(* IEC 61131-3 sources: eCockpitGit/test_project/src/%F%00 Library/%F%Common Functions/%F%Conversion/%F%Array/%F%BOOL Array, 4 files *)

(* ---- %POU%FU_BoolArrayToDWord.st ---- *)
//This functions converts an array of bools to a word, a maximum of 32 bools can be converted
//It must be used in the following way
//FU_BoolArrayToDWord(pArray:= ADR(BoolArray), usiSize:= SIZEOF(BoolArray));
// |**Version**|**Author**| **Date** |**Changes**
// | 1         | NSN      | 28-03-18 | Creation
// | 1.1       | NSN      | 13-06-18 | Updated names and types
FUNCTION FU_BoolArrayToDWord : DWORD
VAR_INPUT
	pArray			:POINTER TO BOOL;	//Address of bool array
	usiSize			:USINT;				//Size of bool array
END_VAR
VAR
	i				:BYTE;
END_VAR
(*%!%__DELIMITER__%!%*)
IF NOT(usiSize = 0) THEN		//Array must be bigger than 0
	IF usiSize > 32 THEN		//Array must be 32 bools or less
		usiSize				:=		32;
	END_IF
	FOR i := 0 TO usiSize - 1 DO
		FU_dwBitSet(dbVar:=FU_BoolArrayToDWord,bIndex:=i,xVal:=pArray^);
		pArray				:=		pArray + 1;
	END_FOR
END_IF

(* ---- %POU%FU_BoolArrayToWord.st ---- *)
//This functions converts an array of bools to a word, a maximum of 16 bools can be converted
//It must be used in the following way
//FU_BoolArrayToWord(pArray:= ADR(BoolArray), usiSize:= SIZEOF(BoolArray));
// |**Version**|**Author**| **Date** |**Changes**
// | 1         | NSN      | 08-03-18 | Creation
// | 1.1       | NSN      | 13-06-18 | Updated names and types
FUNCTION FU_BoolArrayToWord : WORD
VAR_INPUT
	pArray			:POINTER TO BOOL;	//Address of bool array
	usiSize			:USINT;				//Size of bool array
END_VAR
VAR
	i				:BYTE;
END_VAR
(*%!%__DELIMITER__%!%*)
IF NOT(usiSize = 0) THEN		//Array must be bigger than 0
	IF usiSize > 16 THEN		//Array must be 16 bools or less
		usiSize					:=		16;
	END_IF
	FOR i := 0 TO usiSize - 1 DO
		FU_wBitSet(bVar:=FU_BoolArrayToWord,bIndex:=i,xVal:=pArray^);
		pArray				:=		pArray + 1;
	END_FOR
END_IF

(* ---- %POU%FU_DWordToBoolArray.st ---- *)
//This functions converts a word value to a bool array
//It must be used in the following way
//FU_DWordToBoolArray(dwIn:=InputWord,pArray:= ADR(BoolArray), usiSize:= SIZEOF(BoolArray));
// |**Version**|**Author**| **Date** |**Changes**
// | 1         | NSN      | 09-03-18 | Creation
// | 1.1       | NSN      | 13-06-18 | Updated names and types
FUNCTION FU_DWordToBoolArray : BOOL
VAR_INPUT
	dwIn			:DWORD;				//Input value
	pArray			:POINTER TO BOOL;	//Address of bool array
	usiSize			:USINT;				//Size of bool array
END_VAR
VAR
	i				:BYTE;
END_VAR
(*%!%__DELIMITER__%!%*)
IF NOT(usiSize = 0) THEN		//Array must be bigger than 0
	IF usiSize > 32 THEN		//Array must be 32 bools or less
		usiSize				:=		32;
	END_IF
	FOR i := 0 TO usiSize - 1 DO
		pArray^				:=		FU_dwBitGet(dbVar:=dwIn,bIndex:=i);
		pArray				:=		pArray + 1;
	END_FOR
END_IF

(* ---- %POU%FU_WordToBoolArray.st ---- *)
//This functions converts a word value to a bool array
//It must be used in the following way
//FU_WordToBoolArray(wIn:=InputWord,pArray:= ADR(BoolArray), usiSize:= SIZEOF(BoolArray));
// |**Version**|**Author**| **Date** |**Changes**
// | 1         | NSN      | 09-03-18 | Creation
// | 1.1       | NSN      | 13-06-18 | Updated names and types
FUNCTION FU_WordToBoolArray : BOOL
VAR_INPUT
	wIn				:WORD;				//Input value
	pArray			:POINTER TO BOOL;	//Address of bool array
	usiSize			:USINT;				//Size of bool array
END_VAR
VAR
	i				:BYTE;
END_VAR
(*%!%__DELIMITER__%!%*)
IF NOT(usiSize = 0) THEN		//Array must be bigger than 0
	IF usiSize > 16 THEN		//Array must be 16 bools or less
		usiSize				:=		16;
	END_IF
	FOR i := 0 TO usiSize - 1 DO
		pArray^				:=		FU_wBitGet(wVar:=wIn,bIndex:=i);
		pArray				:=		pArray + 1;
	END_FOR
END_IF
